TYPE udt_FixXX_Persistent_Input :
STRUCT

	Prod_Ref_Time:						UINT;
	Prod_Target:							UINT;

END_STRUCT
END_TYPE

(* stored: Version 1.1.0.1, ProductVersion 3.1.4024.5
   DUT udt_FixXX_Persistent_Input: Id {1f6596ad-59a2-4256-8723-07c85b664c75} *)
